(*These are axis parameters that are set up during commissioning and
in theory don't neeed to be change as part of daily moving of axes.
For instance they may be changed due to poor parameter selection
or change of instrument configuration.*)
TYPE ST_AxisConfig :
STRUCT
    //Axis Parameters
    fOverride: LREAL := 100; //Controller override (%). Acts as a global velocity scaling factor for the axis. Default: 100%
    fHomePosition: LREAL := 0; //Position to set the axis to after completing the homing sequence
    fHomeFinishDistance: LREAL := 0; //Distance to move back into the working zone after homing is complete
    eHomeSeq: E_HomingRoutines; //Homing sequence routine to execute
    bRestorePosition: BOOL := TRUE; //Option to restore the position or not during a shutdown
    bEnableStopWithAnyLimitSwitch: BOOL := TRUE; //Option to stop the axis when either the forward or backward limit switch is triggered

    //Advanced homing parameters
    stHomingConfig: ST_HomingConfig; //Configuration for advanced homing routines

    //Backlash compensation config
    stBacklashConfig: ST_BacklashConfig; //Settings for managing backlash compensation

    // CoE
    stCoEParameters : ST_AxisCoE;

    //Temperature disable configuration
    bEnableTemperatureDisable: BOOL := FALSE; //Enable axis disabling due to high temperature
    fMaxTemperature: REAL := 0.0; //Maximum temperature allowed before disabling
    fTempScalingFactor: REAL := 10.0; //Scaling factor for temperature readings

    // Use external brake / airpad
    stAirpadBrake: ST_AirpadBrakeConfig;
    bAirpadManualControl: BOOL := FALSE; //Allow manual control airpad

    // Configure automatic enable / disable
    bAutoEnable: BOOL := FALSE; //Automatically enable an axis when issuing a motion command
    bAutoDisable: BOOL := FALSE; //Automatically disable an axis when motion completed/stopped
    tAutoDisableHysteresis: TIME := T#3S; //Hystersis before issuing automatic disable command after motion completed/stopped

    tCommandHandlerTimeout: TIME := T#15S; //Note: Should be larger than required timeouts for airpad and external brake.
    nCommandHandlerWaitCycles: UINT := 1; //Number of cycles to wait after permits are ready before releasing command to NC. Prevents 4358/4223 errors.

    //Read and Write parameters
    eAxisParameters: E_AxisParameters; //Enumeration of axis parameters for read/write operations
    fWriteAxisParameter: LREAL; //Value to write to the selected axis parameter
    fReadAxisParameter: LREAL; //Current value of the selected axis parameter
    fWriteMinSoftLimit: LREAL; //Value to write minimum position soft limit
    fWriteMaxSoftLimit: LREAL; //Value to write maximum position soft limit

    //Multi-master axis parameters
    astMultiMasterAxis: ARRAY [1..4] OF ST_GearAxis; //Master axes for multi-master configuration
    astMultiMasterAxisLatched: ARRAY [1..4] OF ST_GearAxis; //A kind of readback since one doesn't exist in AXIS_REF
    afMultiSlaveAxisRatio: ARRAY [1..GVL_APP.nAXIS_NUM] OF LREAL; //Slave axis ratios for multi-master setup
    anMultiSlaveAxisIndex: ARRAY [1..2] OF UINT; // These are the slit slave axes, which need to be geared in

    // Read only MC parameters
    bReadMcParametersValid: BOOL:= FALSE; //Indicates validity of MC parameter readings
    bReadMcParametersError: BOOL:= FALSE; //Indicates error in MC parameter readings
    fVelocityDefaultSlow: LREAL; //Read only - AxisManualVelocitySlow
    fVelocityDefaultFast: LREAL; //Read only - AxisManualVelocityFast
    fHomingVelToCam: LREAL; //Read only - AxisVelocityToCam
    fHomingVelFromCam: LREAL; //Read only - AxisVelocityFromCam
    fVeloMax: LREAL; //Read only - AxisMaxVelocity
    fMaxAcc: LREAL; //Read only - AxisMaximumAcceleration
    fMaxDec: LREAL; //Read only - AxisMaximumDeceleration
    fDefaultAcc: LREAL; //Read only - AxisDefaultAcceleration
    fDefaultDec: LREAL; //Read only - AxisDefaultDeceleration
    bEnMinSoftPosLimit: BOOL; //Read only - EnableLimitForward
    fMinSoftPosLimit: LREAL; //Read only - SWLimitForward
    bEnMaxSoftPosLimit: BOOL; //Read only - EnableLimitBackward
    fMaxSoftPosLimit: LREAL; //Read only - SWLimitBackward
    bEnPositionLagMonitoring: BOOL; //Read only - EnablePositionLagMonitoring
    fMaxPosLagValue: LREAL; //Read only - MaxPositionLag
    bEnTargetPositionMonitoring: BOOL; //Read only - AxisEnTargetPositionMonitoring
    fTargetPositionWindow: LREAL; //Read only - AxisTargetPositionWindow
    fAxisEncoderScalingNumerator: LREAL := 0.0; //Read only
    fAxisEncoderScalingDenominator: LREAL := 0.0; //Read only
    stDriveInfo: ST_DriveInfo; //Drive info to e.g. deduce if current axis is connected to Sercos interface
END_STRUCT
END_TYPE

(* stored: Version 1.1.0.1
   DUT ST_AxisConfig: Id {e00fe310-8ff8-452a-800a-823efa83b1a3} *)
